{attribute addProperty BoxType "EK1122-0000-0018"}
{attribute addProperty Id "Beckhoff_EL33xxsub_EK1100EK1100_179A0949162"}
{attribute addProperty CRC "2957642324"}
{attribute addProperty SizeInBites "16"}
{attribute addProperty SizeInBytes "2"}
TYPE Beckhoff_EL33xxEK1122_B04A0A54 EXTENDS EK1122_179A0949 :
STRUCT
	{attribute addProperty Name "Beckhoff_EL33xxsub_EK1100"}
	Beckhoff_EL33xxsub_EK1100 : EK1100_179A0949;
END_STRUCT
END_TYPE

(* stored: Version 1.2.0.0, ProductVersion 3.1.4024.9
   DUT Beckhoff_EL33xxEK1122_B04A0A54: Id {a3f61bd5-2077-4755-adcb-4a9bb1b0b0a5} *)
